PROGRAM MAIN
VAR
END_VAR

END_PROGRAM

(* stored: Version 1.1.0.1
   POU MAIN: Id {3e909943-f812-42e2-9d48-d0aa2efabea3} *)
